(* IEC 61131-3 sources: collections/src/Fifo, 4 files *)

(* ---- IFifo.st ---- *)
NAMESPACE Simatic.Ax.Collections
    INTERFACE IFifo
        METHOD Enqueue : IListItem
            VAR_INPUT
                item : IListItem;
            END_VAR
        END_METHOD

        METHOD Dequeue : IListItem
        END_METHOD

        METHOD Count : INT
        END_METHOD

    END_INTERFACE
END_NAMESPACE

(* ---- IStack.st ---- *)
NAMESPACE Siemens.Ax.Collections
    INTERFACE IFifo
        METHOD Write
            VAR_INPUT
                item : IListItem;
            END_VAR
        END_METHOD
        METHOD Read : IListItem
        END_METHOD
        METHOD Count : INT END_METHOD
    END_INTERFACE
END_NAMESPACE

(* ---- Fifo.st ---- *)
NAMESPACE Simatic.Ax.Collections
    CLASS Fifo IMPLEMENTS IFifo
        VAR PRIVATE
            _list : LinkedList;
        END_VAR

        METHOD PUBLIC FINAL Enqueue : IListItem
            VAR_INPUT
                item : IListItem;
            END_VAR

            Enqueue := _list.Add(item := item);
        END_METHOD

        METHOD PUBLIC Dequeue : IListItem
            Dequeue := _list.Tail();
            _list.Remove(_list.Tail());
        END_METHOD

        METHOD PUBLIC Count : INT
            Count := _list.Count();
        END_METHOD
END_CLASS

END_NAMESPACE

(* ---- Stack.st ---- *)
NAMESPACE Siemens.Ax.Collections
    CLASS Stack IMPLEMENTS IStack
        VAR PRIVATE
            _list : LinkedList;
        END_VAR

        METHOD PUBLIC FINAL Push : IListItem
            VAR_INPUT
                item : IListItem;
            END_VAR

            _list.Add(item := item);
        END_METHOD

        METHOD PUBLIC Pop : IListItem
            Pop := _list.Head();
            _list.Remove(_list.Head());
        END_METHOD

        METHOD PUBLIC Count : INT
            Count := _list.Count();
        END_METHOD

        METHOD PUBLIC Top : IListItem
            Top := _list.Head();
        END_METHOD
END_CLASS

END_NAMESPACE
